TYPE "KukaRobot_UserOutput_1"
VERSION : 0.1
   STRUCT
      Public : Struct
         GO_CurrentMode : USInt;
         GO_CurrentPartType : USInt;
         GO_SpeedActual : USInt;
         GO_RobotTaskSequence : Byte;
         GO5_RobGrip1Status : Byte;
         GO6_RobGrip2Status : Byte;
         GO7 : Byte;
         GO8 : Byte;
         GO9 : Byte;
         GO10 : Byte;
      END_STRUCT;
      Gripper : Struct
         DO129_Grip1GoWork : Bool;
         DO130_Grip1GoHome : Bool;
         DO131_Grip2GoWork : Bool;
         DO132_Grip2GoHome : Bool;
         DO133 : Bool;
         DO134 : Bool;
         DO135 : Bool;
         DO136 : Bool;
         DO137 : Bool;
         DO138 : Bool;
         DO139 : Bool;
         DO140 : Bool;
         DO141 : Bool;
         DO142 : Bool;
         DO143 : Bool;
         DO144 : Bool;
         DO145 : Bool;
         DO146 : Bool;
         DO147 : Bool;
         DO148 : Bool;
         DO149 : Bool;
         DO150 : Bool;
         DO151 : Bool;
         DO152 : Bool;
         DO153 : Bool;
         DO154 : Bool;
         DO155 : Bool;
         DO156 : Bool;
         DO157 : Bool;
         DO158 : Bool;
         DO159 : Bool;
         DO160 : Bool;
      END_STRUCT;
      Home : Struct
         DO161_WaitForHomeSeqStart : Bool;
         DO162_GoHomeFail : Bool;
         DO163_HomeSeqOK : Bool;
         DO164_WaitForAutoStart : Bool;
         DO165_AutoCycle : Bool;
         DO166 : Bool;
         DO167 : Bool;
         DO168 : Bool;
         DO169 : Bool;
         DO170 : Bool;
         DO171 : Bool;
         DO172 : Bool;
         DO173 : Bool;
         DO174 : Bool;
         DO175 : Bool;
         DO176 : Bool;
         DO177_PressPut1Area : Bool;
         DO178_PressPut2Area : Bool;
         DO179_GlueArea : Bool;
         DO180_Robot2Area : Bool;
         DO181 : Bool;
         DO182 : Bool;
         DO183 : Bool;
         DO184 : Bool;
         DO185 : Bool;
         DO186 : Bool;
         DO187 : Bool;
         DO188 : Bool;
         DO189 : Bool;
         DO190 : Bool;
         DO191 : Bool;
         DO192 : Bool;
      END_STRUCT;
      Special : Struct
         DO193 : Bool;
         DO194 : Bool;
         DO195 : Bool;
         DO196 : Bool;
         DO197 : Bool;
         DO198 : Bool;
         DO199 : Bool;
         DO200 : Bool;
         DO201 : Bool;
         DO202 : Bool;
         DO203 : Bool;
         DO204 : Bool;
         DO205 : Bool;
         DO206 : Bool;
         DO207 : Bool;
         DO208 : Bool;
         DO209 : Bool;
         DO210 : Bool;
         DO211 : Bool;
         DO212 : Bool;
         DO213 : Bool;
         DO214 : Bool;
         DO215 : Bool;
         DO216 : Bool;
         DO217 : Bool;
         DO218 : Bool;
         DO219 : Bool;
         DO220 : Bool;
         DO221 : Bool;
         DO222 : Bool;
         DO223 : Bool;
         DO224 : Bool;
      END_STRUCT;
      Cycle : Struct
         DO225_ScanPosInside : Bool;
         DO226_ScanPos1Reach : Bool;
         DO227_ScanPos2Reach : Bool;
         DO228_ScanPos3Reach : Bool;
         DO229_ScanPos4Reach : Bool;
         DO230_ScanPos5Reach : Bool;
         DO231_ScanPos6Reach : Bool;
         DO232_ScanPos7Reach : Bool;
         DO233_ScanPoseFinish : Bool;
         DO234 : Bool;
         DO235 : Bool;
         DO236 : Bool;
         DO237 : Bool;
         DO238 : Bool;
         DO239 : Bool;
         DO240 : Bool;
         DO241_SPalletPickInside : Bool;   // Shaft取料过程中
         DO242_SPalletPickFinish : Bool;   // Shaft取料完成
         DO243_SPalletPickFull : Bool;   // Shaft料盘取空
         "DO244_" : Bool;
         "DO245_" : Bool;
         "DO246_" : Bool;
         "DO247_" : Bool;
         "DO248_" : Bool;
         DO249_ShaftScanPutInside : Bool;   // Shaft读码工位放料过程中
         DO250_ShaftScanPutFinish : Bool;   // Shaft读码工位放料完成
         "DO251_" : Bool;
         "DO252_" : Bool;
         DO253_SScanPickInside : Bool;   // Shaft读码工位取料过程中
         DO254_SScanPickFinish : Bool;   // Shaft读码工位取料完成
         "DO255_" : Bool;
         "DO256_" : Bool;
         DO257_TablePickInside : Bool;   // 转台Ring取料过程中  2#区域  小转台
         DO258_TablePickFinish : Bool;   // 转台Ring取料完成
         "DO259_" : Bool;
         "DO260_" : Bool;
         DO261_RingScanInside : Bool;   // Ring扫码过程中
         DO262_RingScanFinish : Bool;   // Ring扫码完成
         DO263_RingScanReach : Bool;   // Ring扫码到位信号
         "DO264_" : Bool;
         DO265_LoadNGInside : Bool;
         DO266_LoadNGFinish : Bool;
         "DO267_" : Bool;
         "DO268_" : Bool;
         "DO269_" : Bool;
         "DO270_" : Bool;
         "DO271_" : Bool;
         "DO272_" : Bool;
         DO273_PressShaftPutInside : Bool;   // Shaft压机放料过程中
         DO274_PressShaftPutFinish : Bool;   // Shaft压机放料完成
         "DO275_" : Bool;
         "DO276_" : Bool;
         DO277_PressRingPutInside : Bool;   // Ring压机放料过程中
         DO278_PressRingPutFinish : Bool;   // Ring压机放料完成
         DO279_Press2Reach : Bool;   // 机器人到达压机上方放料位置
         "DO280_" : Bool;
         DO281_PressPickInside : Bool;   // 压机取料过程中
         DO282_PressPickFinish : Bool;   // 压机取料完成
         "DO283_" : Bool;
         "DO284_" : Bool;
         "DO285_" : Bool;
         "DO286_" : Bool;
         "DO287_" : Bool;
         "DO288_" : Bool;
         DO289_GluePutInside : Bool;   // 点胶放料过程中
         DO290_GluePutFinish : Bool;   // 点胶放料完成
         DO291 : Bool;
         DO292 : Bool;
         DO293 : Bool;
         DO294 : Bool;
         DO295 : Bool;
         DO296 : Bool;
         DO297_MaintainInside : Bool;
         DO298_MaintainFinish : Bool;
         DO299 : Bool;
         DO300_HomeInside : Bool;
         DO301_HomeFinish : Bool;
         DO302 : Bool;
         DO303 : Bool;
         DO304 : Bool;
         DO305_GripScanInside : Bool;
         DO306_GripScanFinish : Bool;
         DO307_ScanPos1Reach : Bool;
         DO308_ScanPos2Reach : Bool;
         DO309_ScanPos3Reach : Bool;
         DO310_ScanPos4Reach : Bool;
         DO311 : Bool;
         DO312 : Bool;
         DO313 : Bool;
         DO314 : Bool;
         DO315 : Bool;
         DO316 : Bool;
         DO317 : Bool;
         DO318 : Bool;
         DO319 : Bool;
         DO320 : Bool;
         DO321 : Bool;
         DO322 : Bool;
         DO323 : Bool;
         DO324 : Bool;
         DO325 : Bool;
         DO326 : Bool;
         DO327 : Bool;
         DO328 : Bool;
         DO329 : Bool;
         DO330 : Bool;
         DO331 : Bool;
         DO332 : Bool;
         DO333 : Bool;
         DO334 : Bool;
         DO335 : Bool;
         DO336 : Bool;
         DO337 : Bool;
         DO338 : Bool;
         DO339 : Bool;
         DO340 : Bool;
         DO341 : Bool;
         DO342 : Bool;
         DO343 : Bool;
         DO344 : Bool;
         DO345 : Bool;
         DO346 : Bool;
         DO347 : Bool;
         DO348 : Bool;
         DO349 : Bool;
         DO350 : Bool;
         DO351 : Bool;
         DO352 : Bool;
         DO353 : Bool;
         DO354 : Bool;
         DO355 : Bool;
         DO356 : Bool;
         DO357 : Bool;
         DO358 : Bool;
         DO359 : Bool;
         DO360 : Bool;
         DO361 : Bool;
         DO362 : Bool;
         DO363 : Bool;
         DO364 : Bool;
         DO365 : Bool;
         DO366 : Bool;
         DO367 : Bool;
         DO368 : Bool;
         DO369 : Bool;
         DO370 : Bool;
         DO371 : Bool;
         DO372 : Bool;
         DO373 : Bool;
         DO374 : Bool;
         DO375 : Bool;
         DO376 : Bool;
         DO377 : Bool;
         DO378 : Bool;
         DO379 : Bool;
         DO380 : Bool;
         DO381 : Bool;
         DO382 : Bool;
         DO383 : Bool;
         DO384 : Bool;
         DO385 : Bool;
         DO386 : Bool;
         DO387 : Bool;
         DO388 : Bool;
         DO389 : Bool;
         DO390 : Bool;
         DO391 : Bool;
         DO392 : Bool;
         DO393 : Bool;
         DO394 : Bool;
         DO395 : Bool;
         DO396 : Bool;
         DO397 : Bool;
         DO398 : Bool;
         DO399 : Bool;
         DO400 : Bool;
         DO401 : Bool;
         DO402 : Bool;
         DO403 : Bool;
         DO404 : Bool;
         DO405 : Bool;
         DO406 : Bool;
         DO407 : Bool;
         DO408 : Bool;
         DO409 : Bool;
         DO410 : Bool;
         DO411 : Bool;
         DO412 : Bool;
         DO413 : Bool;
         DO414 : Bool;
         DO415 : Bool;
         DO416 : Bool;
      END_STRUCT;
      Safety : Struct
         DO417 : Bool;
         DO418 : Bool;
         DO419 : Bool;
         DO420 : Bool;
         DO421 : Bool;
         DO422 : Bool;
         DO423 : Bool;
         DO424 : Bool;
         DO425 : Bool;
         DO426 : Bool;
         DO427 : Bool;
         DO428 : Bool;
         DO429 : Bool;
         DO430 : Bool;
         DO431 : Bool;
         DO432 : Bool;
         DO433 : Bool;
         DO434 : Bool;
         DO435 : Bool;
         DO436 : Bool;
         DO437 : Bool;
         DO438 : Bool;
         DO439 : Bool;
         DO440 : Bool;
         DO441 : Bool;
         DO442 : Bool;
         DO443 : Bool;
         DO444 : Bool;
         DO445 : Bool;
         DO446 : Bool;
         DO447 : Bool;
         DO448 : Bool;
         DO449 : Bool;
         DO450 : Bool;
         DO451 : Bool;
         DO452 : Bool;
         DO453 : Bool;
         DO454 : Bool;
         DO455 : Bool;
         DO456 : Bool;
         DO457 : Bool;
         DO458 : Bool;
         DO459 : Bool;
         DO460 : Bool;
         DO461 : Bool;
         DO462 : Bool;
         DO463 : Bool;
         DO464 : Bool;
         DO465 : Bool;
         DO466 : Bool;
         DO467 : Bool;
         DO468 : Bool;
         DO469 : Bool;
         DO470 : Bool;
         DO471 : Bool;
         DO472 : Bool;
         DO473 : Bool;
         DO474 : Bool;
         DO475 : Bool;
         DO476 : Bool;
         DO477 : Bool;
         DO478 : Bool;
         DO479 : Bool;
         DO480 : Bool;
         DO481 : Bool;
         DO482 : Bool;
         DO483 : Bool;
         DO484 : Bool;
         DO485 : Bool;
         DO486 : Bool;
         DO487 : Bool;
         DO488 : Bool;
         DO489 : Bool;
         DO490 : Bool;
         DO491 : Bool;
         DO492 : Bool;
         DO493 : Bool;
         DO494 : Bool;
         DO495 : Bool;
         DO496 : Bool;
         DO497 : Bool;
         DO498 : Bool;
         DO499 : Bool;
         DO500 : Bool;
         DO501 : Bool;
         DO502 : Bool;
         DO503 : Bool;
         DO504 : Bool;
         DO505 : Bool;
         DO506 : Bool;
         DO507 : Bool;
         DO508 : Bool;
         DO509 : Bool;
         DO510 : Bool;
         DO511 : Bool;
         DO512 : Bool;
      END_STRUCT;
   END_STRUCT;

END_TYPE

